# EPICS autosave request: iocs/usb-2408-ioc/auto_settings.req
# Settings restored at the next start of usb-2408-ioc.
# Ported from upstream USB2408_settings.req and the per-template
# measComp*_settings.req files it includes, minus the records this port does
# not have (Ao Return/Pulse, Ao SyncMaster, Ai Rate).
#
# Macros: P (record prefix)

$(P)PollSleepMS

$(P)AiMode

$(P)Ai1Range
$(P)Ai1Type
$(P)Ai2Range
$(P)Ai2Type
$(P)Ai3Range
$(P)Ai3Type
$(P)Ai4Range
$(P)Ai4Type
$(P)Ai5Range
$(P)Ai5Type
$(P)Ai6Range
$(P)Ai6Type
$(P)Ai7Range
$(P)Ai7Type
$(P)Ai8Range
$(P)Ai8Type

$(P)Ti1Scale
$(P)Ti1TCType
$(P)Ti1OpenTCDetect
$(P)Ti1Filter
$(P)Ti2Scale
$(P)Ti2TCType
$(P)Ti2OpenTCDetect
$(P)Ti2Filter
$(P)Ti3Scale
$(P)Ti3TCType
$(P)Ti3OpenTCDetect
$(P)Ti3Filter
$(P)Ti4Scale
$(P)Ti4TCType
$(P)Ti4OpenTCDetect
$(P)Ti4Filter
$(P)Ti5Scale
$(P)Ti5TCType
$(P)Ti5OpenTCDetect
$(P)Ti5Filter
$(P)Ti6Scale
$(P)Ti6TCType
$(P)Ti6OpenTCDetect
$(P)Ti6Filter
$(P)Ti7Scale
$(P)Ti7TCType
$(P)Ti7OpenTCDetect
$(P)Ti7Filter
$(P)Ti8Scale
$(P)Ti8TCType
$(P)Ti8OpenTCDetect
$(P)Ti8Filter

$(P)Ao1Range
$(P)Ao1TweakVal
$(P)Ao1SyncEnable
$(P)Ao2Range
$(P)Ao2TweakVal
$(P)Ao2SyncEnable

$(P)WaveDigNumPoints
$(P)WaveDigFirstChan
$(P)WaveDigNumChans
$(P)WaveDigDwell
$(P)WaveDigExtTrigger
$(P)WaveDigExtClock
$(P)WaveDigContinuous
$(P)WaveDigAutoRestart
$(P)WaveDigRetrigger
$(P)WaveDigTriggerCount
$(P)WaveDigBurstMode
$(P)WaveDigReadWF.SCAN

$(P)WaveGenUserNumPoints
$(P)WaveGenIntNumPoints
$(P)WaveGenUserDwell
$(P)WaveGenIntDwell
$(P)WaveGenExtTrigger
$(P)WaveGenExtClock
$(P)WaveGenContinuous
$(P)WaveGenRetrigger
$(P)WaveGenTriggerCount

$(P)WaveGen1Enable
$(P)WaveGen1WaveType
$(P)WaveGen1PulseWidth
$(P)WaveGen1PulseDelay
$(P)WaveGen1Amplitude
$(P)WaveGen1Offset
$(P)WaveGen2Enable
$(P)WaveGen2WaveType
$(P)WaveGen2PulseWidth
$(P)WaveGen2PulseDelay
$(P)WaveGen2Amplitude
$(P)WaveGen2Offset
